FUNCTION derivcvar_M_HardwareMap_t: LREAL
VAR_INPUT
    state: STATE;
END_VAR

derivcvar_M_HardwareMap_t := 1.0;

END_FUNCTION

(* stored: ProductVersion 3.1.0.18, Version 1.1.0.1 *)
